TYPE TcoEq2Transfer_Status EXTENDS TcoCore.TcoStruct:
STRUCT


		ActionDescription:STRING;
		
END_STRUCT
END_TYPE

(* stored: Version 1.1.0.1
   DUT TcoEq2Transfer_Status: Id {e757431f-2392-4391-9c28-3ef50a6f7d1a} *)
